Staubli VAL3: getOnline.pgx

public program getOnline(num x_nCamID (dimensions=1), bool& x_bOnlineState[] (dimensions=1))
  local bool l_bError
begin
  //-----------------------------------------------------------------------
  //Header begin
  //Description of program
  //  Returns the Online state of the In-Sight sensor.
  //
  //Input parameters
  //  num x_nCamID :
  //    role : camera's ID
  //
  //Output parameters
  //  bool x_bOnlineState :
  //    role : mode  of camera
  //    possible values : true  -> The In-Sight sensor is currently Online
  //                      false -> The In-Sight sensor is currently Offline
  //Examples
  //
  //
  //History
  //  Creation : 19-05-08 - f.Rob
  //Header end
  //-----------------------------------------------------------------------

  nProgram[x_nCamID]=3
  call sendCommand(x_nCamID,"GO",l_bError)
  x_bOnlineState=true
  //No errors
  if !l_bError
    //The In-Sight sensor is currently Online
    if cCamera[x_nCamID].nErrorCode==21
      x_bOnlineState=true
    else
      //The In-Sight sensor is currently Offline
      x_bOnlineState=false
    endIf
  else
    x_bOnlineState=false
  endIf
end
